TYPE E_ReactDrive :
(
	Clamp := 1,
	CoverHoriz := 2,
	CoverVerti := 3,
	CoverBoth := 4,
	Complete
)USINT;
END_TYPE

(* stored: Version 1.1.0.1, ProductVersion 3.1.0.25
   DUT E_ReactDrive: Id {c5a8efbd-5f95-4126-ad3e-38f2d3135146} *)
